// TIA Portal V16 export
// export: Created 2021-11-12T13:31:58.2133824Z, ExportSetting WithDefaults, DisplayName Totally Integrated Automation Portal, DisplayVersion V16 Update 3, DisplayName TIA Portal Version Control Interface, DisplayVersion V16 Update 2, DisplayName TIA Portal Openness, DisplayVersion V16 Update 3, DisplayName SINAMICS Startdrive Advanced, DisplayVersion V16 Update 5, DisplayName SINAMICS Startdrive G130, G150, S120, S150, SINAMICS MV, S210, DisplayVersion V16 Update 5, DisplayName SINAMICS Startdrive G110M, G120, G120C, G120D, G120P, G115D, DisplayVersion V16 Update 5, DisplayName STEP 7 Professional, DisplayVersion V16 Update 3, DisplayName STEP 7 Safety, DisplayVersion V16, DisplayName WinCC UA Professional, DisplayVersion V16 Update 3
DATA_BLOCK "STATUS_Zone000"   // DB176
{ S7_Optimized_Access := 'TRUE'; DB_Accessible_From_OPC_UA := 'FALSE' }
VERSION : 0.1
// stored: AutoNumber true, DBAccessibleFromOPCUA false, IsOnlyStoredInLoadMemory false, IsRetainMemResEnabled false, IsWriteProtectedInAS false, MemoryReserve 100
   VAR
      Zone000_Mode : Struct   // Status of zone 000
         Main : "UDT_Status_main";
         Specific : "UDT_Zone_Status_specific";
         Error : "UDT_Error01";
      END_STRUCT;
      StationMEM1_Mode : Struct   // Status of station MEM1
         Main : "UDT_Status_main";
         Specific : "UDT_Zone_Status_specific";
         Error : "UDT_Error01";
      END_STRUCT;
      xxxxx___BinarySensors___xxxxx_1 : Byte;
      "EQ01-BL01" : Bool;   // Hladinový snímač Min LSL 1513 Čerpací jímka 2 (15m3)
      "EQ01-BL02" : Bool;   // Hladinový snímač Max LSH 1514 Čerpací jímka 2 (15m3)
      "EQ01-BL03" : Bool;   // Hladinový snímač Min LSL 1515 Čerpací jímka 3 (5m3)
      "EQ01-BL04" : Bool;   // Hladinový snímač Max LSH 1516 Čerpací jímka 3 (5m3)
      xxxxx___Drives___xxxxx_1 : Byte;
      "EQ01-MA01" : Struct   // Pump (P51) / Čerpadlo cirkulace (P31)
         Main : "UDT_Status_main";
         Specific : "UDT_Drive1_Status_specific";
         Error : "UDT_Error01";
      END_STRUCT;
      "EQ01-MA02" : Struct   // Pump (P52) / Valve with servomotor (A1417) - draining
         Main { S7_SetPoint := 'True'} : "UDT_Status_main";
         Specific { S7_SetPoint := 'True'} : "UDT_Drive1_Status_specific";
         Error { S7_SetPoint := 'True'} : "UDT_Error01";
      END_STRUCT;
      "EQ02-MA01" : Struct   // Pump (P61) / Valve with servomotor (A1417) - draining
         Main { S7_SetPoint := 'True'} : "UDT_Status_main";
         Specific { S7_SetPoint := 'True'} : "UDT_Drive1_Status_specific";
         Error { S7_SetPoint := 'True'} : "UDT_Error01";
      END_STRUCT;
      "UC11-TA01" : Struct   // Frequence inverter for P51 / Frekvenční měnič ( pro P33)
         Main { S7_SetPoint := 'True'} : "UDT_Status_main";
         Specific { S7_SetPoint := 'True'} : "UDT_SINAMICS_G120_Status_specific";
         Error { S7_SetPoint := 'True'} : "UDT_Error02";
      END_STRUCT;
      "UC11-TA02" : Struct   // Frequence inverter for P52 / Frekvenční měnič
         Main { S7_SetPoint := 'True'} : "UDT_Status_main";
         Specific { S7_SetPoint := 'True'} : "UDT_SINAMICS_G120_Status_specific";
         Error { S7_SetPoint := 'True'} : "UDT_Error02";
      END_STRUCT;
      "UC11-TA03" : Struct   // Frequence inverter for P61 / Frekvenční měnič
         Main { S7_SetPoint := 'True'} : "UDT_Status_main";
         Specific { S7_SetPoint := 'True'} : "UDT_SINAMICS_G120_Status_specific";
         Error { S7_SetPoint := 'True'} : "UDT_Error02";
      END_STRUCT;
      xxxxx__Alarms__xxxxx : Byte;
      ArchivePeriodicallyBufferWarning : Struct   // Periodicall buffer archive is almoust full / Periodická vyrovnávací paměť je téměř plná.
         Main { S7_SetPoint := 'True'} : "UDT_Status_main";
         Specific { S7_SetPoint := 'True'} : "UDT_DI_Mon_Status_specific";
         Error { S7_SetPoint := 'True'} : "UDT_Error01";
      END_STRUCT;
      ArchivePeriodicallyBufferAlarm : Struct   // Periodicall buffer archive is full / Periodická vyrovnávací paměť je plná.
         Main { S7_SetPoint := 'True'} : "UDT_Status_main";
         Specific { S7_SetPoint := 'True'} : "UDT_DI_Mon_Status_specific";
         Error { S7_SetPoint := 'True'} : "UDT_Error01";
      END_STRUCT;
      ArchiveItemBufferWarning : Struct   // Item buffer archive is almoust full / Neperiodická vyrovnávací paměť je téměř plná.
         Main { S7_SetPoint := 'True'} : "UDT_Status_main";
         Specific { S7_SetPoint := 'True'} : "UDT_DI_Mon_Status_specific";
         Error { S7_SetPoint := 'True'} : "UDT_Error01";
      END_STRUCT;
      ArchiveItemBufferAlarm : Struct   // Item buffer archive is full / Neperiodická vyrovnávací paměť je plná.
         Main { S7_SetPoint := 'True'} : "UDT_Status_main";
         Specific { S7_SetPoint := 'True'} : "UDT_DI_Mon_Status_specific";
         Error { S7_SetPoint := 'True'} : "UDT_Error01";
      END_STRUCT;
   END_VAR
BEGIN
END_DATA_BLOCK
